# EPICS substitutions: src/makeBaseApp/top/pcdsMotorApp/Db/archive__APPNAME_.substitutions
#
# _APPNAME_ substitutions file
#

# Generate iocAdmin archive request
#	Macros:
#		IOC		- PV prefix for all iocAdmin PV's
# Typically, IOC will be expanded in the iocBoot/<ioc_name>/Makefile
file archive_iocAdmin.template
{
	{
		# Hack till msi supports empty substitutions
		IOC		=	$(IOC)
	}
}

# Generate autosave Save/Restore status archive requests
#	Macros:
#		IOC		- PV prefix for all IOC autosave Save/Restore PV's
# Typically, IOC will be expanded in the iocBoot/<ioc_name>/Makefile
file archive_SR.template
{
	{
		# Hack till msi supports empty substitutions
		IOC		=	$(IOC)
	}
}

# Generate EVR archive request
#	Macros:
#		EVR		- PV prefix for all EVR PV's
# Typically, EVR will be expanded in the iocBoot/<ioc_name>/Makefile
file archive_evr.template
{
	{
		# Hack till msi supports empty substitutions
		IOC		=	$(IOC),
		EVR		=	$(EVR)
	}
}
